{attribute 'qualified_only'}
VAR_GLOBAL CONSTANT
  MAX_STACKSIZE : DINT := 32000*10;
END_VAR

(* stored: Version 1.1.0.1, ProductVersion 3.1.4020.12
   GVL ProfilerParameterList: Id {1e8f260f-5e09-45f9-a5ed-a85e826c75c5}, ParameterList True *)
